// SIMATIC S7-200 SMART project (STEP 7-Micro/WIN SMART), CPU ST60

SYMBOL_TABLE 系统符号
Always_On        SM0.0    // 始终接通
END_SYMBOL_TABLE

ORGANIZATION_BLOCK MAIN:OB1
TITLE=程序注释
BEGIN
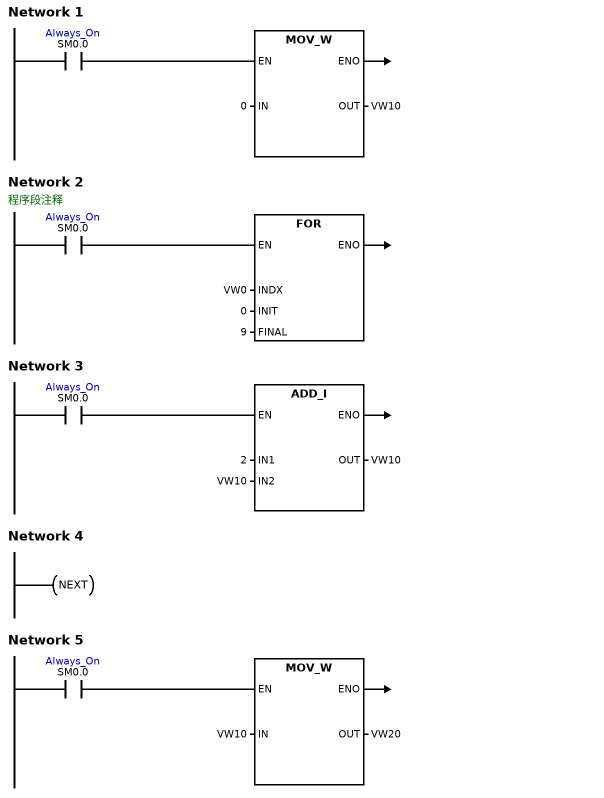
Network 1
LD     Always_On:SM0.0
MOVW   0, VW10
Network 2
// 程序段注释
LD     Always_On:SM0.0
FOR    VW0, 0, 9
Network 3
LD     Always_On:SM0.0
+I     2, VW10
Network 4
NEXT
Network 5
LD     Always_On:SM0.0
MOVW   VW10, VW20
END_ORGANIZATION_BLOCK
